// TIA Portal V18 export
DATA_BLOCK "H-8_DB"   // DB78
VERSION : 0.1
// stored: AutoNumber true, DBAccessibleFromOPCUA true, DBAccessibleFromWebserver true, InstanceOfName PIDNormal_FB_1.0, InstanceOfType FB
"PIDNormal_FB_1.0"
   // VAR_INPUT
   //    PV : Real;
   //    ResetPID : Bool;
   //    SetP1 : Bool;
   //    SetP2 : Bool;
   //    SetP3 : Bool;
   //    SetP4 : Bool;
   //    SetP5 : Bool;
   //    ManExt : Bool;
   //    Scale : Bool;
   // END_VAR
   // VAR_OUTPUT
   //    Out_word : Word;
   // END_VAR
   // VAR_IN_OUT
   //    Data : "PID_DT";
   // END_VAR
   // VAR
   //    IEC_Timer_0 : IEC_TIMER;
   //    "Last Time" : Time;
   //    IEC_Timer_1 : IEC_TIMER;
   //    DeltaTimeR : Real;
   //    "Always On" : Bool;
   //    ER : Real;
   //    Last_ER : Real;
   //    LMN_P : Real;
   //    LMN_I : Real;
   //    LMN_D : Real;
   //    LMN_AUTO : Real;
   //    LMN : Real;
   //    SP1 : Real;
   //    SP2 : Real;
   //    Gain : Real;
   //    Ti : Time;
   //    Td : Time;
   //    Tm_lag : Time;
   //    Man_ON : Bool;
   //    MAN : Real;
   //    LMN_HI : Real;
   //    LMN_LO : Real;
   //    Reset : Bool;
   //    ResetHMI : Bool;
   //    SPAKt : Real;
   //    SP3 : Real;
   //    SP4 : Real;
   //    SP5 : Real;
   // END_VAR
BEGIN
END_DATA_BLOCK
